/// Additional axis IO (direct linked) for AX5xxx axis.
TYPE ST_AxisIO :
STRUCT
	stIn 	AT %I* 	:ST_AxisIn;
	stOut	AT %Q* 	:ST_AxisOut;
END_STRUCT
END_TYPE

(* stored: Version 1.1.0.1, ProductVersion 3.1.4020.12
   DUT ST_AxisIO: Id {3b7e3fad-6baa-4128-8ea8-0a9cc00677f8} *)
